{attribute addProperty BoxType "EP9128-0021-0016"}
{attribute addProperty Id "A_0007_EP9128_0021_0017A_0007_EP9128_0021_0017_0A93B5694598574.75A_0004_EP9128_0021_0016_2_EP9128_1021EP9128_179A0949162"}
{attribute addProperty CRC "3082329405"}
{attribute addProperty SizeInBites "4614"}
{attribute addProperty SizeInBytes "576.75"}
TYPE A_0004_EP9128_0021_0016_B7B89D3D EXTENDS EP9128_179A0949 :
STRUCT
	{attribute addProperty Name "A_0007_EP9128_0021_0017"}
	A_0007_EP9128_0021_0017 : A_0007_EP9128_0021_0017_0A93B569;
	{attribute addProperty Name "A_0004_EP9128_0021_0016_2_EP9128_1021"}
	A_0004_EP9128_0021_0016_2_EP9128_1021 : EP9128_179A0949;
END_STRUCT
END_TYPE

(* stored: Version 1.2.0.0, ProductVersion 3.1.4024.9
   DUT A_0004_EP9128_0021_0016_B7B89D3D: Id {8d6cfe31-2aa9-45d3-9ab8-9abe96dc406c} *)
